FUNCTION F_Log
VAR_INPUT
	value : T_MaxString;
END_VAR

Tc2_System.ADSLOGSTR(0, value, '%');

END_FUNCTION

(* stored: Version 1.1.0.1
   POU F_Log: Id {3282e1c6-2408-4fe0-a2ef-9039b76e2bfe}, SpecialFunc None *)
